// SIMATIC S7-200 SMART project (STEP 7-Micro/WIN SMART), CPU ST30

SYMBOL_TABLE Table 1
V_VB             VB0
END_SYMBOL_TABLE

SYMBOL_TABLE System Symbols
Clock_1s         SM0.5    // Clock pulse that is ON for 0.5 s, OFF for 0.5 s, for a duty cycle time of 1 s.
END_SYMBOL_TABLE

ORGANIZATION_BLOCK MAIN:OB1
TITLE=Program Comments
BEGIN
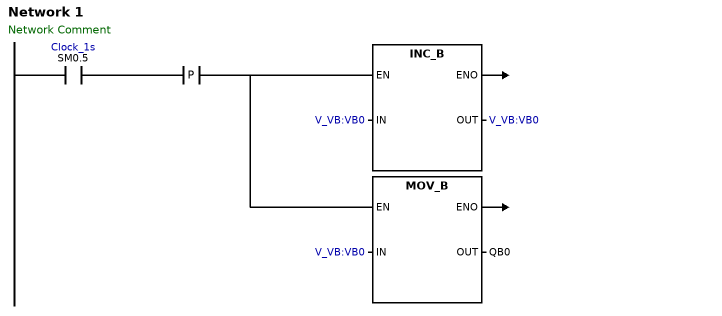
Network 1
// Network Comment
// (network saved uncompiled; LAD cells follow)
// row 0: c0 -| |- Clock_1s:SM0.5  c1 -|P|-  v  c2 --  c3 [INC_B EN:=power@row0, IN:=V_VB:VB0, ENO=>power, OUT=>V_VB:VB0]  c4 ->
// row 1: c1 ^v  c3 [box]
// row 2: c1 ^  c2 --  c3 [MOV_B EN:=power@row2, IN:=V_VB:VB0, ENO=>power, OUT=>QB0]  c4 ->
// row 3: c3 [box]
END_ORGANIZATION_BLOCK

DATA_BLOCK_TAB Page_1
BEGIN
//DATA PAGE COMMENTS
//Press F1 for help and example data page
         V_VB, 2
END_DATA_BLOCK_TAB
